{attribute 'qualified_only'}
{attribute 'strict'}
TYPE E_ActWorkUnits :
(
	eActWork_Idle		:=	0,
	eActWork_ApronSlide	:=  1,
	eActWork_ApronFold	:=  2,
	eActWork_BackGauge	:=  3,
	eActWork_Clamp		:=  4,
	eActWork_Slitter	:=  5
) DINT;
END_TYPE

(* stored: Version 1.1.0.1, ProductVersion 3.1.4024.12
   DUT E_ActWorkUnits: Id {1eb5b629-e91b-426c-9707-016aa7dc65d6} *)
